// TIA Portal V18 export
DATA_BLOCK "Global data"   // DB2
{ S7_Optimized_Access := 'TRUE' }
VERSION : 0.1
// stored: AutoNumber true, DBAccessibleFromOPCUA true, IsOnlyStoredInLoadMemory false, IsRetainMemResEnabled false, IsWriteProtectedInAS false, MemoryReserve 100
   VAR
      data1 : Bool;
      data2 : Bool;
      data3 : Bool;
      data4 : Bool;
      data5 : Bool;
      data6 : Bool;
      data7 : Bool;
      data8 : Bool;
   END_VAR
   VAR RETAIN
      dataB1 : Byte := 10;
   END_VAR
   VAR
      dataB2 : Byte := 10;
      dataB3 : Byte := 10;
      dataB4 : Byte := 10;
      dataW1 : Word := 10;
   END_VAR
   VAR RETAIN
      dataW2 : Word := 20;
      dataW3 : Word := 20;
      dataW4 : Word := 20;
   END_VAR
   VAR
      dataW5 : Word := 20;
   END_VAR
BEGIN
END_DATA_BLOCK
